(* Logix 5000 project; controller SS1 Emulate 5570 rev 33.11; software revision 33.00 *)

TASK MainTask (continuous, watchdog 500 ms) : MainProgram

MODULES
   Local : Emulate 5570 (ICP 2, rev 33.11)
       : 1756-IB16 (ICP 3, rev 3.1, Input RPI 20 ms)
       : 1756-OB16D (ICP 4, rev 3.1, Output RPI 20 ms)
END_MODULES

PROGRAM MainProgram   (* main routine TextRoutine *)

ROUTINE TextRoutine   (* structured text *)
   
   
END_ROUTINE
END_PROGRAM
